PROGRAM CarTrafficLight
VAR
	StartTrafficLightTimer: BOOL := FALSE;
	DelayPedestrianLight: TIME;
	TimerTrafficLight: TON;
END_VAR

IF GVL.ButtonPedestrian AND NOT StartTrafficLightTimer THEN
	TimerTrafficLight( IN := GVL.ButtonPedestrian, PT := T#10S );
	StartTrafficLightTimer := TRUE;
	
ELSIF StartTrafficLightTimer AND TimerTrafficLight THEN
	IF GVL.CarLightGreen THEN
		GVL.CarLightGreen := FALSE;
		GVL.CarLightYellow := TRUE;
	ELSIF GVL.CarLightYellow THEN
		GVL.CarLightYellow := FALSE;
		GVL.CarLightRed:= TRUE;	
	END_IF

StartTrafficLightTimer := FALSE;
GVL.ButtonPedestrian := FALSE;	
END_IF

END_PROGRAM

(* stored: Version 1.1.0.1, ProductVersion 3.1.4024.12
   POU CarTrafficLight: Id {937bb74f-8fa3-4ea3-85e7-c63a585c47b5}, SpecialFunc None *)
